FUNCTION_BLOCK FB_WS
VAR_INPUT
END_VAR
VAR_OUTPUT
END_VAR
VAR
	KL_Wetterstation_group_0_0_1		: EIB_GROUP_ADDR := (MAIN:=0, SUB_MAIN:=0, NUMBER:=1);
	Wetterstation_Lesen			 		: FB_WS_Input;

END_VAR

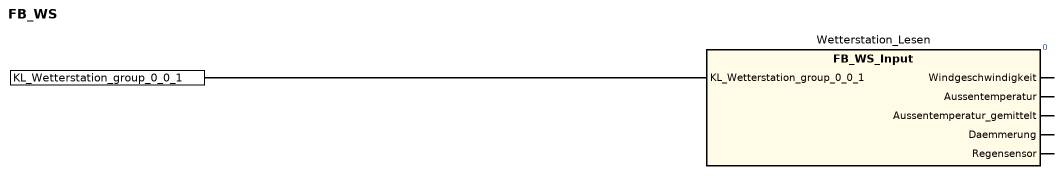
Wetterstation_Lesen(KL_Wetterstation_group_0_0_1 := KL_Wetterstation_group_0_0_1); // FB_WS_Input

END_FUNCTION_BLOCK

(* stored: Version 1.1.0.1, ProductVersion 3.1.4024.9
   POU FB_WS: Id {86159f38-bf79-4e5b-adb9-b4ce76416872}, SpecialFunc None *)
